{attribute 'no_check'}
//Returns the count of a particular char found in a string line
FUNCTION getCntCharInStr : INT
VAR_INPUT
	Chars													:	STRING(5):=';';
	Strline													:	T_MaxString;
END_VAR             										
VAR                 
	tmpString												:	T_MaxString ;										
	pos,k													:	INT;
END_VAR

IF StrLine <> '' AND Chars <> ''
THEN
	MEMSET(ADR(tmpString),0,SIZEOF(tmpString));
	MEMCPY(ADR(tmpString),ADR(Strline),TO_UDINT(LEN(Strline)));
	pos 													:= FIND (tmpString,Chars);
	WHILE pos <> 0 DO	
		k													:=  pos + (LEN(Chars) - 1);
		tmpString											:=	RIGHT(tmpString,LEN(tmpString) - k);
		pos 												:= 	FIND (tmpString,Chars);
		getCntCharInStr										:=	getCntCharInStr+1;
	END_WHILE;
ELSE
	getCntCharInStr											:= 0;
END_IF

END_FUNCTION

(* stored: Version 1.1.0.1, ProductVersion 3.1.4024.13
   POU getCntCharInStr: Id {f492d5fa-af5e-4452-9cce-6f54509917fe}, SpecialFunc None *)
